PROGRAM MAIN
VAR
END_VAR

(*CALL POUs*)
	WaterTankFilling();
	HMI();

END_PROGRAM

(* stored: Version 1.1.0.1, ProductVersion 3.1.4024.15
   POU MAIN: Id {0622d039-adf9-47cb-91cc-f67f7f72f49e}, SpecialFunc None *)
